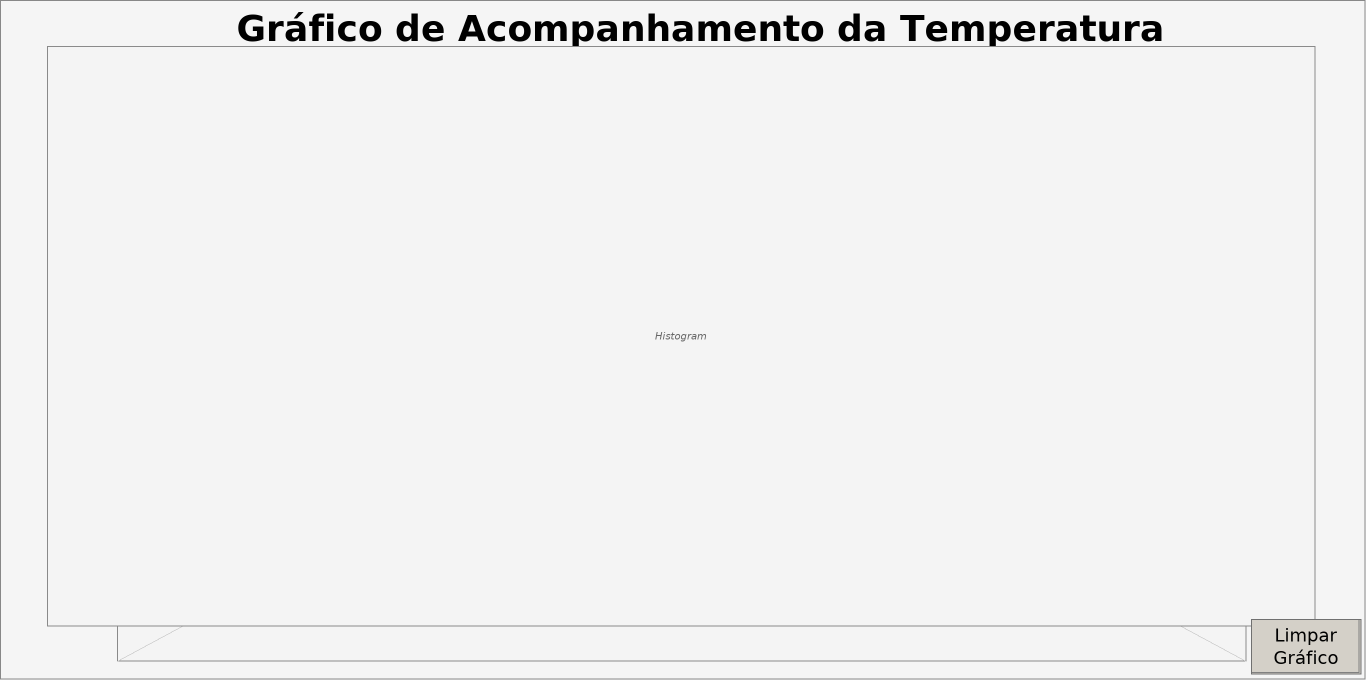
VISUALIZATION Grafico_2  // 1366x680
    Image (117,52 1129x609), image: ImagePool.Screenshot_3
    Histogram (47,46 1268x580), scale format: %.1f, scale 0..150
        p1518820177: GVL_P.arrTempVisu020
        p102497268: GVL_P.arrTempVisu020
        p788070771: ARRAY [1..720] OF REAL
    Label (262,7 877x43), "Gráfico de Acompanhamento da Temperatura"
    Histogram (47,46 1268x580), scale format: %.1f, scale 0..150
        p1518820177: GVL_P.arrTemp020
        p102497268: GVL_P.arrTemp020
        p788070771: ARRAY [1..720] OF REAL
    Button (1251,619 110x55), "Limpar Gráfico"
        OnMouseClick: execute {
            FOR gvl.i:=0 TO 720 BY 1 DO
            	gvl_p.arrTemp020[gvl.i]:= 0;
            	gvl_p.arrTempVisu020[gvl.i]:= 0;
            	END_FOR
        }
END_VISUALIZATION

(* stored: Version 1.1.0.1, ProductVersion 3.1.4024.12
   Visu Grafico_2: Id {6fbf8b98-0a47-4fda-bebc-650f6e070dee} *)
